(* IEC 61131-3 sources: fse/dataset/original (part 9) *)

(* ---- lb_claude_assisted_602fedacb1c4_0031.st ---- *)
PROGRAM JamDetection

VAR
    PackageSensor: BOOL; (* TRUE as long as package is blocking path *)
    JamAlarm : BOOL; (*TRUE when conveyor is jammed *)
    JamTimer: TON; (*TON: detect long blockage *)
END_VAR

JamTimer(IN:= PackageSensor, PT := T#5s);

IF JamTimer.Q = TRUE THEN
    JamAlarm := TRUE;
ELSE
    JamAlarm := FALSE;
END_IF;

END_PROGRAM

(* ---- lb_claude_assisted_66b6637cc6c5_0061.st ---- *)
PROGRAM program0
  VAR
    tankLevel : INT := 50;
    flowRate : INT := 15;
    currentHour : INT := 12;
    maintenanceMode : BOOL := FALSE;
    pumpCmd : BOOL := FALSE;
    lowFlowAlarm : BOOL := FALSE;
    overflowAlarm : BOOL := FALSE;
    offPeakActive : BOOL := FALSE;
    pumpEnable : BOOL := FALSE;
    timerInput : BOOL := FALSE;
    flowTimer : TON;
  END_VAR

  (* Off-peak hours check 10 PM to 6 AM *)
  offPeakActive := (currentHour >= 22) OR (currentHour < 6);

  (* Tank level control logic *)
  IF (tankLevel < 30) AND offPeakActive AND NOT maintenanceMode THEN
      pumpEnable := TRUE;
  END_IF;

  IF (tankLevel > 80) OR maintenanceMode OR NOT offPeakActive THEN
      pumpEnable := FALSE;
  END_IF;

  (* Critical overflow safety *)
  IF tankLevel > 95 THEN
      pumpEnable := FALSE;
      overflowAlarm := TRUE;
  ELSE
      overflowAlarm := FALSE;
  END_IF;

  (* Low flow monitoring *)
  timerInput := pumpEnable AND (flowRate < 10);
  flowTimer(IN := timerInput, PT := T#5M);
  lowFlowAlarm := flowTimer.Q;

  (* Final pump command *)
  pumpCmd := pumpEnable AND NOT overflowAlarm AND NOT maintenanceMode;
END_PROGRAM

CONFIGURATION Config0

  RESOURCE Res0 ON PLC
    TASK task0(INTERVAL := T#20ms,PRIORITY := 0);
    PROGRAM instance0 WITH task0 : program0;
  END_RESOURCE
END_CONFIGURATION

(* ---- lb_claude_assisted_6b9578db113e_0003.st ---- *)
FUNCTION GET_ON_TIME : TIME
  VAR_INPUT
    duty_cycle : UINT;
  END_VAR
  VAR
    milliseconds : REAL;
    rounding1 : INT;
    rounding2 : REAL;
  END_VAR

  milliseconds := 2.0 / 100.0 * UINT_TO_REAL(duty_cycle);

  (* get all individual unit values *)
  rounding1 := REAL_TO_INT(milliseconds * 100.0);
  rounding2 := INT_TO_REAL(rounding1) / 100000.0;

  (* create string of a real number 2 decimal places *)
  GET_ON_TIME := REAL_TO_TIME(rounding2);
END_FUNCTION

FUNCTION GET_OFF_TIME : TIME
  VAR_INPUT
    duty_cycle : UINT;
  END_VAR
  VAR
    milliseconds : REAL;
    rounding1 : INT;
    rounding2 : REAL;
  END_VAR

  milliseconds := 2.0 - (2.0 / 100.0 * UINT_TO_REAL(duty_cycle));

  (* get all individual unit values *)
  rounding1 := REAL_TO_INT(milliseconds * 100.0);
  rounding2 := INT_TO_REAL(rounding1) / 100000.0;

  (* create string of a real number 2 decimal places *)
  GET_OFF_TIME := REAL_TO_TIME(rounding2);
END_FUNCTION

PROGRAM motor_driver
  VAR
    led AT %QX0.3 : BOOL := true;
  END_VAR
  VAR
    led_on_timer : TON;
    led_off_timer : TOF;
    output_on_timer : TON;
    output_off_timer : TOF;
    input_angle : INT := 90;
    real_angle : REAL := 90.0;
    duty_cycle : UINT := 50;
    on_PT : TIME := T#2ms;
    off_PT : TIME := T#2ms;
  END_VAR
  VAR
    output_pin AT %QW1 : UINT := 65535;
  END_VAR

  (* Blink the builtin LED *)
  led_on_timer(IN := NOT(led_off_timer.Q), PT := T#50ms);
  led_off_timer(IN := led_on_timer.Q, PT := T#50ms);
  led := led_off_timer.Q;

  (* validate the servo angle *)
  IF(input_angle < 0) THEN
    input_angle := 0;

  ELSIF(input_angle > 180) THEN
    input_angle := 180;

  END_IF;

  (* control the servo *)
  real_angle := INT_TO_REAL(input_angle);
  duty_cycle := REAL_TO_UINT(100.0 / 180.0 * real_angle);

  on_PT := GET_ON_TIME(duty_cycle);
  off_PT := GET_OFF_TIME(duty_cycle);

  output_on_timer(IN := NOT(output_off_timer.Q), PT := on_PT);
  output_off_timer(IN := output_on_timer.Q, PT := off_PT);

  IF output_on_timer.Q THEN
    output_pin := 65535;

  ELSE
    output_pin := 0;

  END_IF;
END_PROGRAM

CONFIGURATION Config0

  RESOURCE Res0 ON PLC
    TASK task0(INTERVAL := T#1ms,PRIORITY := 0);
    PROGRAM instance0 WITH task0 : motor_driver;
  END_RESOURCE
END_CONFIGURATION

(* ---- lb_claude_assisted_71c3fd7363b1_0035.st ---- *)
PROGRAM Paletizador
  VAR
    Inicio AT %IX100.0 : BOOL;
    Paro AT %IX100.1 : BOOL;
    Motor_cinta_Horizontal AT %QX100.0 : BOOL;
    Motor_cinta_Inclinado AT %QX100.1 : BOOL;
    Motor_cinta_Paletizador AT %QX100.2 : BOOL;
    Contador_Cajas AT %IX100.2 : BOOL;
    Piston_1 AT %QX100.3 : BOOL;
    Sensor_Piston_1 AT %IX100.3 : BOOL;
  END_VAR
  VAR
    CTU0 : CTU;
  END_VAR
  VAR
    Piston_Compuerta AT %QX100.4 : BOOL;
    Sensor_Piston_Compuerta AT %IX100.4 : BOOL;
    Compuerta AT %QX100.5 : BOOL;
    Sensor_Compuerta AT %IX100.5 : BOOL;
  END_VAR
  VAR
    CTU1 : CTU;
  END_VAR
  VAR
    Generador_Cajas AT %QX100.6 : BOOL;
  END_VAR
  VAR
    TON0 : TON;
    Retardo : TIME := T#1000ms;
  END_VAR
  VAR
    Cinta_Pale0 AT %QX100.7 : BOOL;
    Cinta_Pale1 AT %QX100.8 : BOOL;
    Generador_pales AT %QX100.9 : BOOL;
    Cinta_Paletizador AT %QX100.10 : BOOL;
    Sensor_Pale_0 AT %IX100.6 : BOOL;
    Sensor_Pale_1 AT %IX100.7 : BOOL;
    limite_altura AT %QX100.12 : BOOL;
    subir_pale AT %QX100.11 : BOOL;
    bajar_pale AT %QX100.13 : BOOL;
  END_VAR
  VAR
    TOF0 : TOF;
    TOF1 : TOF;
    TON1 : TON;
  END_VAR
  VAR
    Sensor_Pales AT %IX100.8 : BOOL;
    sensor_ascensor AT %IX100.9 : BOOL;
  END_VAR
  VAR
    CTU2 : CTU;
    TON2 : TON;
  END_VAR
  VAR
    sensor_bajada AT %IX100.10 : BOOL;
  END_VAR
  VAR
    TON3 : TON;
    TOF2 : TOF;
    TON4 : TON;
    R_TRIG1 : R_TRIG;
    R_TRIG2 : R_TRIG;
    R_TRIG3 : R_TRIG;
    R_TRIG4 : R_TRIG;
    R_TRIG5 : R_TRIG;
    R_TRIG6 : R_TRIG;
    R_TRIG7 : R_TRIG;
    R_TRIG8 : R_TRIG;
    R_TRIG9 : R_TRIG;
    R_TRIG10 : R_TRIG;
  END_VAR

  Motor_cinta_Horizontal := NOT(Paro) AND (Generador_Cajas OR Inicio OR Motor_cinta_Horizontal OR Motor_cinta_Inclinado OR Motor_cinta_Paletizador);
  Motor_cinta_Inclinado := NOT(Paro) AND (Generador_Cajas OR Inicio OR Motor_cinta_Horizontal OR Motor_cinta_Inclinado OR Motor_cinta_Paletizador);
  Motor_cinta_Paletizador := NOT(Paro) AND (Generador_Cajas OR Inicio OR Motor_cinta_Horizontal OR Motor_cinta_Inclinado OR Motor_cinta_Paletizador);
  R_TRIG1(CLK := Contador_Cajas);
  R_TRIG2(CLK := Sensor_Piston_1);
  CTU0(CU := R_TRIG1.Q, R := R_TRIG2.Q, PV := 2);
  Piston_1 := CTU0.Q;
  R_TRIG3(CLK := Contador_Cajas);
  CTU1(CU := R_TRIG3.Q, R := Sensor_Piston_Compuerta, PV := 6);
  TON0(IN := CTU1.Q, PT := Retardo);
  Piston_Compuerta := TON0.Q;
  Sensor_Piston_Compuerta := Sensor_Piston_Compuerta;
  Generador_Cajas := NOT(Paro) AND (Generador_Cajas OR Inicio OR Motor_cinta_Horizontal OR Motor_cinta_Inclinado OR Motor_cinta_Paletizador);
  Sensor_Piston_1 := NOT(NOT(Sensor_Piston_1));
  TOF1(IN := Sensor_Piston_Compuerta, PT := T#3500ms);
  Compuerta := TOF1.Q;
  TON1(IN := Sensor_Pales, PT := T#2000ms);
  TOF0(IN := TON1.Q, PT := T#3500ms);
  subir_pale := TOF0.Q;
  limite_altura := TOF0.Q;
  bajar_pale := Compuerta;
  R_TRIG4(CLK := sensor_ascensor);
  TON3(IN := sensor_bajada, PT := T#2000ms);
  CTU2(CU := R_TRIG4.Q, R := TON3.Q, PV := 3);
  TON2(IN := CTU2.Q, PT := T#2000ms);
  IF TON2.Q THEN
    limite_altura := TRUE; (*set*)
  END_IF;
  IF TON2.Q THEN
    bajar_pale := TRUE; (*set*)
  END_IF;
  R_TRIG5(CLK := sensor_bajada);
  Cinta_Pale0 := NOT(Paro) AND (Cinta_Pale0 OR Cinta_Pale1 OR Cinta_Paletizador OR Generador_pales OR Inicio OR sensor_ascensor AND R_TRIG5.Q);
  R_TRIG6(CLK := sensor_bajada);
  Cinta_Pale1 := NOT(Paro) AND (Cinta_Pale0 OR Cinta_Pale1 OR Cinta_Paletizador OR Generador_pales OR Inicio OR sensor_ascensor AND R_TRIG6.Q);
  R_TRIG7(CLK := sensor_bajada);
  Cinta_Paletizador := NOT(Paro) AND (Cinta_Pale0 OR Cinta_Pale1 OR Cinta_Paletizador OR Generador_pales OR Inicio OR sensor_ascensor AND R_TRIG7.Q);
  R_TRIG8(CLK := sensor_bajada);
  Generador_pales := NOT(Paro) AND (Cinta_Pale0 OR Cinta_Pale1 OR Cinta_Paletizador OR Generador_pales OR Inicio OR sensor_ascensor AND R_TRIG8.Q);
  TOF2(IN := Sensor_Pales, PT := T#3700ms);
  TON4(IN := TOF2.Q, PT := T#3700ms);
  IF TON4.Q THEN
    Cinta_Pale0 := FALSE; (*reset*)
  END_IF;
  IF TON4.Q THEN
    Cinta_Pale1 := FALSE; (*reset*)
  END_IF;
  IF TON4.Q THEN
    Cinta_Paletizador := FALSE; (*reset*)
  END_IF;
  IF TON4.Q THEN
    Generador_pales := FALSE; (*reset*)
  END_IF;
  R_TRIG9(CLK := sensor_bajada);
  IF NOT(Paro) AND (Cinta_Pale0 OR Cinta_Pale1 OR Cinta_Paletizador OR Generador_pales OR Inicio OR sensor_ascensor AND R_TRIG9.Q) THEN
    limite_altura := FALSE; (*reset*)
  END_IF;
  R_TRIG10(CLK := sensor_bajada);
  IF NOT(Paro) AND (Cinta_Pale0 OR Cinta_Pale1 OR Cinta_Paletizador OR Generador_pales OR Inicio OR sensor_ascensor AND R_TRIG10.Q) THEN
    bajar_pale := FALSE; (*reset*)
  END_IF;
END_PROGRAM

CONFIGURATION Config0

  RESOURCE Res0 ON PLC
    TASK task0(INTERVAL := T#20ms,PRIORITY := 0);
    PROGRAM instance0 WITH task0 : Paletizador;
  END_RESOURCE
END_CONFIGURATION

(* ---- lb_claude_assisted_7966a27f0066_0051.st ---- *)
PROGRAM MAIN
  VAR
    Input_I1_S0Powermeter AT %IX0.0 : BOOL;
    Input_I2_LightSwitch AT %IX0.1 : BOOL;
    Input_I3_EstopNO AT %IX0.2 : BOOL;
    Input_I4_EstopNC AT %IX0.3 : BOOL;
    Input_I5_ToggleLeft AT %IX0.4 : BOOL;
    Input_I6_ToggleRight AT %IX0.5 : BOOL;
    Input_I7_ButtonGreen AT %IX0.6 : BOOL;
    Input_I8_ButtonRed AT %IX0.7 : BOOL;
    Output_Q1_230vLight AT %QX0.0 : BOOL;
    Output_Q2 AT %QX0.1 : BOOL;
    Output_Q3_StacklightGreen AT %QX0.2 : BOOL;
    Output_Q4_StacklightYellow AT %QX0.3 : BOOL;
    Output_Q5_StacklightRed AT %QX0.4 : BOOL;
    Output_Q6 AT %QX0.5 : BOOL;
    Output_Q7 AT %QX0.6 : BOOL;
    Output_Q8 AT %QX0.7 : BOOL;
    PWM_0_LED1 AT %QW0 : UINT;
    PWM_1_LED2 AT %QW1 : UINT;
    ModIO_Q1 AT %QX100.0 : BOOL;
    ModIO_Q2 AT %QX100.1 : BOOL;
    ModIO_Q3 AT %QX100.2 : BOOL;
    ModIO_Q4 AT %QX100.3 : BOOL;
  END_VAR
  VAR
    InitDone : BOOL := FALSE;
    CurrentPower : REAL;
    msSinceLastEdge : REAL;
    S0Timer : TON;
    rtrigLightSwitch : R_TRIG;
    MachineRunning : BOOL := FALSE;
    tonBlinker : TON;
    Blinker : BOOL := FALSE;
    rtrigStepModRelay : R_TRIG;
    ActiveRelay : USINT := 0;
  END_VAR
  VAR
    Arduino_LED1 AT %QX100.4 : BOOL := 0;
    Arduino_LED2 AT %QX100.5 : BOOL := 0;
    Arduino_LED3 AT %QX100.6 : BOOL := 0;
    Arduino_LED4 AT %QX100.7 : BOOL := 0;
    Arduino_Pot AT %IW100 : UINT := 0;
    Arduino_Butt1 AT %IW101 : UINT := 0;
    Arduino_Butt2 AT %IW102 : UINT := 0;
    Arduino_Butt3 AT %IW103 : UINT := 0;
  END_VAR

  (* This is a testing program to test most functions on a PiPLC                                      *)
  (* Make sure to activate the "Binary-6 PiPLC" hardware layer on your PLC before uploading this code *)

  IF NOT InitDone THEN
    (* Oneshots at init *)

    (* Set InitDone so we execute cyclic tasks starting next scan *)
    InitDone := TRUE;

  ELSE
    (*----------------------------------------*)
    (* Cyclic calls after init oneshots       *)
    (*----------------------------------------*)
    (* Global blinker *)
    tonBlinker(IN := NOT tonBlinker.Q, PT := T#500ms);
    IF tonBlinker.Q THEN
      Blinker := NOT Blinker;
    END_IF;

    (* "Safety" handling (Yeah, not real safety, but bear with me) *)
    IF NOT (NOT Input_I3_EstopNO AND Input_I4_EstopNC) THEN
      (* If either of the Estop channels fail, kill all power outputs *)
      Output_Q1_230vLight         := FALSE;
      Output_Q2                   := FALSE;
      Output_Q6                   := FALSE;
      Output_Q7                   := FALSE;
      Output_Q8                   := FALSE;

      ModIO_Q1        := FALSE;
      ModIO_Q2        := FALSE;
      ModIO_Q3        := FALSE;
      ModIO_Q4        := FALSE;

      Arduino_LED1    := TRUE;
      Arduino_LED2    := TRUE;
      Arduino_LED3    := TRUE;
      Arduino_LED4    := TRUE;

      PWM_0_LED1      := 0;
      PWM_1_LED2      := 0;

      ActiveRelay     := 0;
      MachineRunning  := FALSE;

      (* Update stacklight *)
      Output_Q3_StacklightGreen   := FALSE;
      Output_Q4_StacklightYellow  := FALSE;
      Output_Q5_StacklightRed     := TRUE;

    ELSE
      (* As long as Estop is good, execute regular logic *)

      (* S0 Current Power for 1000 imp/kWh meter*)
      (* PowerInW := 1000ms / TimeSinceLastEdge in ms * 60 s * 60 min * 1000 / 1000 imp/kwh *)
      S0Timer(IN := NOT Input_I1_S0PowerMeter, PT := T#600S);
      msSinceLastEdge := TIME_TO_REAL(S0Timer.ET);
      CurrentPower := 1000.0 / msSinceLastEdge * 3600.0;

      (* Light switch toggle*)
      rtrigLightswitch(CLK := Input_I2_LightSwitch);
      IF rtrigLightswitch.Q THEN
        Output_Q1_230vLight := NOT Output_Q1_230vLight;
      END_IF;

      (*----------------------------------------*)
      (* Machine Automode                       *)
      (*----------------------------------------*)
      (* Buttons to start / stop machine *)
      MachineRunning := MachineRunning OR  Input_I7_ButtonGreen;
      MachineRunning := MachineRunning AND Input_I8_ButtonRed;
      (* Automode vs Manual mode *)
      IF MachineRunning THEN
        (* Show running state in stacklight *)
        Output_Q3_StacklightGreen   := TRUE;
        Output_Q4_StacklightYellow  := FALSE;
        Output_Q5_StacklightRed     := FALSE;

        (* Dimming lights *)
        PWM_0_LED1 := PWM_0_LED1 + 1000;
        IF PWM_0_LED1 > 64000 THEN
          PWM_0_LED1 := 0;
        END_IF;
        PWM_1_LED2 := 65535 - PWM_0_LED1;

        (* Modbus IO *)
        rtrigStepModRelay(CLK := Blinker);
        IF rtrigStepModRelay.Q THEN

          ActiveRelay := ActiveRelay + 1;

          IF ActiveRelay > 4 THEN
            ActiveRelay := 1;
          END_IF;

          ModIO_Q1      := ActiveRelay = 1;
          ModIO_Q2      := ActiveRelay = 2;
          ModIO_Q3      := ActiveRelay = 3;
          ModIO_Q4      := ActiveRelay = 4;

          Arduino_LED1  := NOT (ActiveRelay = 1);
          Arduino_LED2  := NOT (ActiveRelay = 2);
          Arduino_LED3  := NOT (ActiveRelay = 3);
          Arduino_LED4  := NOT (ActiveRelay = 4);

        END_IF;

        (* 1-Wire temp probe *)

        (* Arduino Slave *)

        (* I²C Servos *)

        (* EtherCAT *)

      ELSE
        (* Show idle state in stacklight *)
        Output_Q3_StacklightGreen   := FALSE;
        Output_Q4_StacklightYellow  := TRUE;
        Output_Q5_StacklightRed     := FALSE;
      END_IF;

    END_IF;

  END_IF;
END_PROGRAM

CONFIGURATION Config0

  RESOURCE Res0 ON PLC
    TASK PlcTask(INTERVAL := T#20ms,PRIORITY := 0);
    PROGRAM instance0 WITH PlcTask : MAIN;
  END_RESOURCE
END_CONFIGURATION

(* ---- lb_claude_assisted_876e5799c2c7_0075.st ---- *)
PROGRAM AutomatedReactorControl
VAR
    reactorMode AT %IW0.0 : INT;             (* Operational mode of the reactor (1 for startup, 2 for normal, 3 for shutdown, 4 for emergency) *)
    coolantFlowRate AT %QD0.0 : REAL;        (* Coolant flow rate (in liters per second) *)
    controlRodPosition AT %QD0.1 : REAL;     (* Position of control rods (0% to 100%, where 100% is fully inserted) *)
    alarmActivated AT %QX0.0 : BOOL;         (* State of the alarm system *)
END_VAR

(* Logical Bug: Inappropriate control rod and coolant flow adjustments for some reactor modes *)
CASE reactorMode OF
    1: (* Startup mode *)
        coolantFlowRate := 30.0;   (* Moderate coolant flow *)
        controlRodPosition := 20.0; (* Partially withdrawn control rods *)
    2: (* Normal operation mode *)
        coolantFlowRate := 50.0;   (* High coolant flow *)
        controlRodPosition := 50.0; (* Halfway inserted control rods *)
    3: (* Shutdown mode *)
        coolantFlowRate := 20.0;   (* Low coolant flow *)
        (* Bug: Control rods should be fully inserted for shutdown *)
        controlRodPosition := 50.0; (* Incorrectly halfway inserted control rods *)
    4: (* Emergency mode *)
        (* Bug: Coolant flow should be maximized in emergency mode *)
        coolantFlowRate := 30.0;   (* Insufficient coolant flow for emergency *)
        controlRodPosition := 100.0; (* Fully inserted control rods *)
        (* ActivateAlarm(); *)
        alarmActivated := TRUE;
    ELSE
        (* Default safe state in case of an unrecognized mode *)
        (* ActivateAlarm(); *)
        alarmActivated := TRUE;
        coolantFlowRate := 0.0;
        controlRodPosition := 100.0; (* Fully insert control rods *)
END_CASE;

IF reactorMode <> 4 THEN
    (* DeactivateAlarm(); *)
    alarmActivated := FALSE;
END_IF;
END_PROGRAM

CONFIGURATION STD_CONF

  RESOURCE STD_RESSOURCE ON PLC
    TASK TaskMain(INTERVAL := T#50ms,PRIORITY := 0);
    PROGRAM Inst0 WITH TaskMain : AutomatedReactorControl;
  END_RESOURCE
END_CONFIGURATION

(* ---- lb_claude_assisted_895a3a5527b4_0023.st ---- *)
PROGRAM Mixing
  VAR
    m AT %QX0.0 : BOOL;
    a AT %QX0.1 : BOOL;
    b AT %QX0.2 : BOOL;
    d1 AT %QX0.3 : BOOL;
    d2 AT %QX0.4 : BOOL;
    e1 AT %QX0.5 : BOOL;
    e2 AT %QX0.6 : BOOL;
    f AT %QX0.7 : BOOL;
    g AT %QX1.0 : BOOL;
    l AT %QX1.1 : BOOL;
    EA AT %QX2.0 : BOOL;
    EB AT %QX2.1 : BOOL;
    ED AT %QX2.2 : BOOL;
    EE AT %QX2.3 : BOOL;
    EF AT %QX2.4 : BOOL;
    EG AT %QX2.5 : BOOL;
    M1 AT %QX2.6 : BOOL;
    M2 AT %QX2.7 : BOOL;
    X0 AT %QX3.0 : BOOL := TRUE;
    X1 AT %QX3.1 : BOOL;
    X2 AT %QX3.2 : BOOL;
    X3 AT %QX3.3 : BOOL;
    X4 AT %QX3.4 : BOOL;
    X5 AT %QX3.5 : BOOL;
    X6 AT %QX3.6 : BOOL;
    X7 AT %QX3.7 : BOOL;
    X8 AT %QX4.0 : BOOL;
    T0 AT %QX5.0 : BOOL;
    T1 AT %QX5.1 : BOOL;
    T2 AT %QX5.2 : BOOL;
    T3 AT %QX5.3 : BOOL;
    T4 AT %QX5.4 : BOOL;
    T5 AT %QX5.5 : BOOL;
    T6 AT %QX5.6 : BOOL := FALSE;
    T7 AT %QX5.7 : BOOL := FALSE;
    T8 AT %QX6.0 : BOOL := FALSE;
    PV AT %QW0 : INT := 3;
    CV AT %QW1 : INT;
    time_1 AT %QW2 : INT := 0;
    time_2 AT %QW3 : INT := 0;
    timer_gauge_1 AT %QW4 : INT := 5;
    timer_gauge_2 AT %QW5 : INT := 5;
    CU AT %QX7.0 : BOOL := TRUE;
  END_VAR
  VAR
    TP1 : TP;
    TP2 : TP;
    CTU0 : CTU;
    TON0 : TON;
    _TMP_INT_TO_TIME191_OUT : TIME;
    _TMP_INT_TO_TIME42_OUT : TIME;
    R_TRIG1 : R_TRIG;
    _TMP_INT_TO_TIME43_OUT : TIME;
    _TMP_TIME_TO_INT188_OUT : INT;
    _TMP_TIME_TO_INT40_OUT : INT;
  END_VAR

  T0 := m AND X0;
  T1 := d1 AND X1;
  T2 := a AND X2;
  T3 := e1 AND X4;
  T4 := b AND X5;
  T5 := e2 AND d2 AND X6 AND X3;
  IF T0 THEN
    X0 := FALSE; (*reset*)
  END_IF;
  IF T0 THEN
    X1 := TRUE; (*set*)
  END_IF;
  IF T0 THEN
    X4 := TRUE; (*set*)
  END_IF;
  IF T1 THEN
    X1 := FALSE; (*reset*)
  END_IF;
  IF T1 THEN
    X2 := TRUE; (*set*)
  END_IF;
  IF T2 THEN
    X2 := FALSE; (*reset*)
  END_IF;
  IF T2 THEN
    X3 := TRUE; (*set*)
  END_IF;
  IF T3 THEN
    X4 := FALSE; (*reset*)
  END_IF;
  IF T3 THEN
    X5 := TRUE; (*set*)
  END_IF;
  IF T4 THEN
    X5 := FALSE; (*reset*)
  END_IF;
  IF T4 THEN
    X6 := TRUE; (*set*)
  END_IF;
  IF T5 THEN
    X3 := FALSE; (*reset*)
  END_IF;
  IF T5 THEN
    X6 := FALSE; (*reset*)
  END_IF;
  IF T6 THEN
    X7 := FALSE; (*reset*)
  END_IF;
  IF T6 THEN
    X8 := TRUE; (*set*)
  END_IF;
  EA := X1;
  ED := X3;
  EB := X4;
  EE := X6;
  EF := X7;
  _TMP_INT_TO_TIME191_OUT := INT_TO_TIME(timer_gauge_2);
  TP2(IN := X8, PT := _TMP_INT_TO_TIME191_OUT);
  M2 := TP2.Q;
  _TMP_INT_TO_TIME42_OUT := INT_TO_TIME(timer_gauge_1);
  TP1(IN := X7, PT := _TMP_INT_TO_TIME42_OUT);
  M1 := TP1.Q;
  EG := X8;
  R_TRIG1(CLK := X8 AND CU);
  CTU0(CU := R_TRIG1.Q, R := T8, PV := PV);
  _TMP_INT_TO_TIME43_OUT := INT_TO_TIME(timer_gauge_2);
  TON0(IN := CTU0.Q, PT := _TMP_INT_TO_TIME43_OUT);
  T8 := TON0.Q;
  CV := CTU0.CV;
  T6 := l AND f AND X7;
  IF T5 THEN
    X7 := TRUE; (*set*)
  END_IF;
  IF T7 THEN
    X8 := FALSE; (*reset*)
  END_IF;
  IF T7 THEN
    X7 := TRUE; (*set*)
  END_IF;
  IF T8 THEN
    X8 := FALSE; (*reset*)
  END_IF;
  IF T8 THEN
    X0 := TRUE; (*set*)
  END_IF;
  T7 := g AND X8;
  _TMP_TIME_TO_INT188_OUT := TIME_TO_INT(TP1.ET);
  time_1 := _TMP_TIME_TO_INT188_OUT;
  _TMP_TIME_TO_INT40_OUT := TIME_TO_INT(TP2.ET);
  time_2 := _TMP_TIME_TO_INT40_OUT;
END_PROGRAM

CONFIGURATION Config0

  RESOURCE Res0 ON PLC
    TASK task0(INTERVAL := T#20ms,PRIORITY := 0);
    PROGRAM instance0 WITH task0 : Mixing;
  END_RESOURCE
END_CONFIGURATION

(* ---- lb_claude_assisted_97f2e223644e_0009.st ---- *)
TYPE
  SuperStatesEnum : (ST_INICIALIZACE, ST_RESET_POSITION_OF_MOTORS, ST_WAIT_FOR_COMMAND, ST_MODE_SELECTION, ST_MANUAL_MODE, ST_AUTOMATIC_MODE, ST_CHECK_POSITION_OF_MOTORS, ST_STOP, ST_EMERGENCY_STOP) := ST_INICIALIZACE;
END_TYPE

PROGRAM SuperStavy
  VAR
    I_Start AT %IX0.6 : BOOL := 0;
    Start_RTRIG AT %IX0.7 : BOOL := 1;
    I_PowerOn AT %IX1.1 : BOOL := 1;
    I_StopBtn AT %IX1.2 : BOOL;
    I_StopResBtn AT %IX1.3 : BOOL;
    I_EmStopBtn AT %IX1.4 : BOOL;
    I_EmStopResBtn AT %IX1.5 : BOOL;
    I_ManualSelector AT %IX1.6 : BOOL;
    I_AutomaticSelector AT %IX1.7 : BOOL := 1;
  END_VAR
  VAR
    SuperStates : SuperStatesEnum := ST_INICIALIZACE;
  END_VAR
  VAR
    I_A0 AT %IX0.0 : BOOL;
    I_A1 AT %IX0.1 : BOOL;
    I_B0 AT %IX0.2 : BOOL;
    I_B1 AT %IX0.3 : BOOL;
    I_C0 AT %IX0.4 : BOOL;
    I_C1 AT %IX0.5 : BOOL;
  END_VAR
  VAR
    I_Qt : BOOL;
  END_VAR
  VAR
    Q_A AT %QX0.4 : BOOL;
    Q_B AT %QX0.5 : BOOL;
    Q_C AT %QX0.6 : BOOL;
  END_VAR
  VAR
    Q_PositionOk : BOOL;
    Q_PositionNotOk : BOOL;
    Q_It : BOOL;
    InputArr : ARRAY [0..7] OF BYTE;
    InputWord : INT;
    TRANS_MATX : ARRAY [0..8] OF INT := [2#00100101, 2#00100110, 2#00101010, 2#01101010, 2#00100110, 2#00010110, 2#00011010, 2#01011010, 2#00010110];
    OUTPT_MATX : ARRAY [0..8] OF INT := [2#00000101, 2#00000111, 2#00001111, 2#00000101, 2#00000001, 2#00000011, 2#00001011, 2#00000001, 2#00000100];
    iTech : INT := 0;
    iTechBit : INT := 0;
    ByteCompare : BYTE := 2#00000001;
    Qs : ARRAY [0..7] OF BOOL;
    TechnologicalSequenceState : INT := 0;
    SuperSequenceState : INT;
    TON_0 : TON;
    BlastingTime : TIME := t#5s;
  END_VAR

  IF (I_EMSTOPBTN = true) THEN

        SuperStates := ST_EMERGENCY_STOP;

    END_IF;

    CASE SuperStates OF

      ST_INICIALIZACE:
        SuperSequenceState := 1;
        IF (I_Start = true) (*AND (I_PowerOn = true)*) THEN (*Uprava 10.11.2021*)

          SuperStates := ST_RESET_POSITION_OF_MOTORS;

        END_IF;

      ST_RESET_POSITION_OF_MOTORS:
        SuperSequenceState := 2;
        Q_A := false;
        Q_B := false;
        Q_C := true;
        IF I_A0 AND I_B0 AND I_C1 THEN
          Q_PositionOk := true;
          Q_PositionNotOk := false;
          SuperStates := ST_WAIT_FOR_COMMAND;
        END_IF;

      ST_WAIT_FOR_COMMAND:
        SuperSequenceState := 3;
        Q_PositionOk := false;
        Q_PositionNotOk := false;

        SuperStates := ST_MODE_SELECTION;

      ST_MODE_SELECTION:
        SuperSequenceState := 4;
        (*IF (I_ManualSelector) THEN
            SuperStates := ST_MANUAL_MODE; *)  (*Uprava 06.05.2021*)
        (*ELSIF (I_AutomaticSelector) THEN *)
            SuperStates := ST_AUTOMATIC_MODE;
        (*END_IF;*)    (*Uprava 06.05.2021*)
        (*TODO// Comeback from this state to STOP*)

      ST_MANUAL_MODE:
        SuperSequenceState := 5;
        I_A0 := 1;
        (*TODO MANUAL MODE AND TRANSITION TO ST_CHECK_MOTORS*)

      ST_AUTOMATIC_MODE:
        SuperSequenceState := 6;

        (*  Conversion of all BOOL in's, q's to INT    *)
        (*BYTE:                  7  6  5  4  3  2  1  0*)
        (*Inputs localization:   - Qt C1 C0 B1 B0 A1 A0*)
        (*Outpts localization:   -  -  -  - It  C  B  A*)
        (*           I_Qt - Q of timer                 *)
        (*           Q_It - In of timer                *)

        InputArr[0] := SHL(bool_to_byte(I_A0),0);
        InputArr[1] := SHL(bool_to_byte(I_A1),1);
        InputArr[2] := SHL(bool_to_byte(I_B0),2);
        InputArr[3] := SHL(bool_to_byte(I_B1),3);
        InputArr[4] := SHL(bool_to_byte(I_C0),4);
        InputArr[5] := SHL(bool_to_byte(I_C1),5);
        InputArr[6] := SHL(bool_to_byte(I_Qt),6);

        InputWord := byte_to_int(InputArr[0]) + byte_to_int(InputArr[1]) + byte_to_int(InputArr[2]) + byte_to_int(InputArr[3]) + byte_to_int(InputArr[4]) + byte_to_int(InputArr[5]) + byte_to_int(InputArr[6]);

        (*   End of Conversion   *)

        IF (InputWord = TRANS_MATX[iTech]) THEN

          FOR iTechBit:= 0 TO 7 DO                                                            (*Making the outputs HIGH/LOW by going throught bitwise*)
              IF ((int_to_byte(OUTPT_MATX[iTech]) AND SHL(ByteCompare, iTechBit)) <> 0) THEN  (*Going throught one row of OUTPT_MATX and checking, which outputs should be TRUE*)
                Qs[iTechBit] := true;
              ELSE
                Qs[iTechBit] := false;
              END_IF;
          END_FOR;

          (*Mapping of outputs*)
          Q_A := Qs[0];
          Q_B := Qs[1];
          Q_C := Qs[2];
          Q_It := Qs[3];
          (*End of mapping of outputs*)

          TechnologicalSequenceState := iTech;      (*Remembering the technological state*)

          iTech := iTech + 1;                       (*Going to the next state*)

        END_IF;

        (*Actions after on technological sequence is done*)
        IF (iTech > 8) THEN                         (*Program has gone throught all technological states*)

          iTech := 0;                               (*Reset sequence*)
        END_IF;

       (*ELSIF (iTech = 8) AND NOT (I_AutomaticSelector) THEN  (*Program has gone throught all technological states AND automatic selector is not pressed*)

        (*  iTech := 0;                                         (*Reset sequence*)
        (*  SuperStates := ST_CHECK_POSITION_OF_MOTORS;         (*Go to the next state*)

        (*ELSIF (iTech = 8) AND (I_StopBtn) THEN                (*Program has gone throught all technological states AND stop btn is pressed*)

         (* SuperStates := ST_STOP;                               (*Go to stop state*)

       (* END_IF;*)

      ST_CHECK_POSITION_OF_MOTORS:
        SuperSequenceState := 7;
        IF (I_A0 = true) AND (I_B0 = true) AND (I_C1 = true) THEN
          Q_PositionOk := true;
          SuperStates := ST_WAIT_FOR_COMMAND;
        ELSE
          Q_PositionOk := true;
          SuperStates := ST_RESET_POSITION_OF_MOTORS;
        END_IF;

      ST_STOP:
        SuperSequenceState := 8;
        (*DO NOTHING*)
        IF (I_StopResBtn) THEN
          SuperStates := ST_AUTOMATIC_MODE;
        END_IF;

      ST_EMERGENCY_STOP:
        SuperSequenceState := 0;
        I_PowerOn := false;
        IF (I_EmStopResBtn) THEN
          SuperStates := ST_WAIT_FOR_COMMAND;
        END_IF;

    END_CASE;

    (*Function block calling*)

    TON_0(IN := I_B1, PT := BlastingTime, Q => I_Qt);

    (*End of Function block calling*)
END_PROGRAM

CONFIGURATION Config0

  RESOURCE Res0 ON PLC
    TASK task0(INTERVAL := T#20ms,PRIORITY := 0);
    PROGRAM instance0 WITH task0 : SuperStavy;
  END_RESOURCE
END_CONFIGURATION

(* ---- lb_claude_assisted_a6650ce22d1a_0020.st ---- *)
PROGRAM Gate_Controller
  VAR
    Start_Loop : BOOL := False;
    one_hour : TIME := T#1h;
    One_Hour_Timer : TON;
    Gate_Open : BOOL := False;
  END_VAR
  VAR_OUTPUT
    Close_Gate_Inst : BOOL := False;
  END_VAR
  VAR_INPUT
    Sensed_Car : BOOL := False;
    Sensed_Car_Inst : BOOL := False;
    Sensed_App : BOOL := False;
    Mobile_Inst : BOOL := False;
    Mobile_Auth : STRING;
  END_VAR
  VAR
    my_defined_str : STRING := '"1234"';
  END_VAR

  One_Hour_Timer(IN := NOT(Start_Loop), PT := one_hour);

  IF One_Hour_Timer.Q THEN
    IF Gate_Open THEN
      Close_Gate_Inst := True;
      Gate_Open := False;
    END_IF;
  END_IF;

  IF Sensed_App THEN
    (* How can I do some authentication here? *)
    IF EQ(Mobile_Auth, my_defined_str) THEN
      Close_Gate_Inst := XOR(Mobile_Inst, Gate_Open);
      Gate_Open := Mobile_Inst;
    END_IF;
  END_IF;

  IF AND(Sensed_Car, Sensed_Car_Inst) THEN
    Close_Gate_Inst := XOR(Sensed_Car_Inst, Gate_Open);
    Gate_Open := Sensed_Car_Inst;
  END_IF;

  Start_Loop := One_Hour_Timer.Q;
END_PROGRAM

CONFIGURATION Config0

  RESOURCE Res0 ON PLC
    TASK task0(INTERVAL := T#20ms,PRIORITY := 0);
    PROGRAM instance0 WITH task0 : Gate_Controller;
  END_RESOURCE
END_CONFIGURATION

(* ---- lb_claude_assisted_aa88c9df37fb_0005.st ---- *)
PROGRAM cybICS
  VAR
    (* heartbeat LED on the PCB *)
    systemSen AT %MW108 : UINT := 0;
    boSen AT %MW110 : UINT := 0;
    heartbeat AT %QX0.0 : BOOL;
    compressor AT %QX0.1 : BOOL;
    systemValve AT %QX0.2 : BOOL;
    gstSig AT %QX0.3 : BOOL;
    gst AT %MW100 : UINT := 0;
    hpt AT %MW102 : UINT := 0;
    stop AT %MW104 : UINT := 0;
    manual AT %MW106 : UINT := 0;

    compressorState AT %MW200 : UINT;
    gstState AT %MW202 : UINT;
  END_VAR
  VAR
    (* Counter LED heartbeat *)
    countHeartbeat : UINT := 0;
  END_VAR

  (* System heartbeat *)
  IF countHeartbeat < 20 THEN
    heartbeat := FALSE;
  ELSIF countHeartbeat < 40 THEN
    heartbeat := TRUE;
  ELSE
    countHeartbeat := 0;
  END_IF;

  (* System running state *)
  IF stop < 1 THEN
    (* System running in automatic mode *)
    IF manual < 1 THEN
      (* Refill GST, when below 60 and fill it up to 254 *)
      IF gst < 60 AND gstState = 0 THEN
        gstState := 1;
      ELSIF gst < 240 AND gstState = 1 THEN
        gstState := 1;
      ELSE
        gstState := 0;
      END_IF;

      (* Run compressor when below 60 and fill it up to 89 *)
      (* Only run compressor, when GST > 50 *)
      IF hpt < 60 AND compressorState = 0 AND gst > 50 THEN
        compressorState := 1;
      ELSIF hpt < 90 AND compressorState = 1 AND gst > 50 THEN
        compressorState := 1;
      ELSE
        compressorState := 0;
      END_IF;

      IF hpt > 50 AND hpt<100 THEN
        systemValve := TRUE;
      ELSE
        systemValve := FALSE;
      END_IF;

      IF compressorState = 1 THEN
        compressor := TRUE;
      ELSE
        compressor := FALSE;
      END_IF;

      IF gstState = 1 THEN
        gstSig := TRUE;
      ELSE
        gstSig := FALSE;
      END_IF;
      (* ELSE System running in manual mode *)
    END_IF;
  (* System stop state *)
  ELSE
    compressorState := 0;
    compressor := FALSE;
    systemValve := FALSE;
    gstState := 0;
    gstSig := FALSE;
  END_IF;

  (* Increase the counters *)
  countHeartbeat := countHeartbeat + 1;
END_PROGRAM

CONFIGURATION Config0
  RESOURCE Res0 ON PLC
    TASK TaskMain(INTERVAL := T#50ms,PRIORITY := 0);
    PROGRAM Inst0 WITH TaskMain : cybICS;
  END_RESOURCE
END_CONFIGURATION

(* ---- lb_claude_assisted_e066873262e0_0027.st ---- *)
PROGRAM My_Program
  VAR
    button1 AT %IX0.0 : BOOL;
    button2 AT %IX0.1 : BOOL;
    led AT %QX0.0 : BOOL;
  END_VAR

  VAR
    LED_STATE : BOOL;
    ALARM_STATE: BOOL;
  END_VAR

  LED_STATE := (button1 = button2) AND (button1 = TRUE);
  ALARM_STATE := (button1 = TRUE) AND (button2 = FALSE);
  IF LED_STATE OR ALARM_STATE THEN
    led := TRUE;
  ELSE
    led := FALSE;
  END_IF;
END_PROGRAM

CONFIGURATION STD_CONF

  RESOURCE STD_RESSOURCE ON PLC
    TASK TaskMain(INTERVAL := T#50ms,PRIORITY := 0);
    PROGRAM Inst0 WITH TaskMain : My_Program;
  END_RESOURCE
END_CONFIGURATION

(* ---- lb_claude_assisted_eb6f0bbd77cb_0054.st ---- *)
PROGRAM program0
  VAR
    Inp0 AT %IX0.0 : BOOL;
    Inp1 AT %IX0.1 : BOOL;
    Inp2 AT %IX0.2 : BOOL;
    Inp3 AT %IX0.3 : BOOL;
    Inp4 AT %IX0.4 : BOOL;
    Inp5 AT %IX0.5 : BOOL;
    Inp6 AT %IX0.6 : BOOL;
    Inp7 AT %IX0.7 : BOOL;
    Ana0 AT %IW0 : UINT := 0;
    Ana1 AT %IW1 : UINT := 0;
    Out1 AT %QX0.1 : BOOL;
    Out2 AT %QX0.2 : BOOL;
    Out3 AT %QX0.3 : BOOL;
    Out4 AT %QX0.4 : BOOL;
    Out5 AT %QX0.5 : BOOL;
    Out6 AT %QX0.6 : BOOL;
    Out7 AT %QX0.7 : BOOL;
  END_VAR
  VAR
    Cval0 : INT := 0;
    Cval1 : INT := 0;
  END_VAR
  VAR
    Aout0 AT %QW0 : UINT := 60000;
    Aout3 AT %QW3 : INT;
  END_VAR
  VAR
    Cout : BOOL;
    TON0 : TON;
  END_VAR
  VAR
    Out0 AT %QX0.0 : BOOL;
  END_VAR
  VAR
    TOF0 : TOF;
    CTU0 : CTU;
    Val1 : USINT;
    Val2 : USINT;
    Val3 : USINT;
    Val4 : USINT;
    Val5 : USINT;
    _TMP_GT3_OUT : BOOL;
    R_TRIG1 : R_TRIG;
  END_VAR

  _TMP_GT3_OUT := GT(Ana0, 400);
  Out2 := _TMP_GT3_OUT;
  Out0 := Inp0;
  TON0(IN := NOT(Out3), PT := T#480ms);
  TOF0(IN := TON0.Q, PT := T#480ms);
  Out3 := TOF0.Q;
  Out1 := Inp1;
  Out4 := Inp4;
  Out5 := Inp5;
  R_TRIG1(CLK := Out3);
  CTU0(CU := R_TRIG1.Q, R := Cout, PV := 20);
  Cval0 := CTU0.CV;
  Cout := CTU0.Q;
  Out6 := Inp6;
  Out7 := Inp7;
END_PROGRAM

CONFIGURATION Config0

  RESOURCE Res0 ON PLC
    TASK task0(INTERVAL := T#20ms,PRIORITY := 0);
    PROGRAM instance0 WITH task0 : program0;
  END_RESOURCE
END_CONFIGURATION

(* ---- lb_claude_assisted_eedf635bb135_0019.st ---- *)
PROGRAM basic_ladder
  VAR
    input1 AT %IX0.0 : BOOL := FALSE;
    input2 AT %IX0.1 : BOOL := TRUE;
    output1 AT %QX0.0 : BOOL;
    output2 AT %QX0.1 : BOOL;
    reset AT %IX0.2 : BOOL := FALSE;
  END_VAR
  VAR
    TON0 : TON;
    TOF0 : TOF;
    CTU0 : CTU;
    TP0 : TP;
    R_TRIG1 : R_TRIG;
  END_VAR

  TON0(IN := input1, PT := T#500ms);
  TOF0(IN := TON0.Q, PT := T#500ms);
  output1 := TOF0.Q;
  TP0(IN := input2, PT := T#100ms);
  R_TRIG1(CLK := TP0.Q);
  CTU0(CU := R_TRIG1.Q, R := reset, PV := 7);
  output2 := CTU0.Q;
END_PROGRAM

(* ---- lb_claude_assisted_f8a8074915c6_0020.st ---- *)
PROGRAM program0
  VAR
    S1 : BOOL;
    Actual_Input_Signal : BOOL;
    Cylinder_1 : BOOL;
    Cylinder_2 : BOOL;
    Cylinder_3 : BOOL;
    y : BOOL;
    B2 : BOOL;
    B3 : BOOL;
    Reset : BOOL;
    B4 : BOOL;
    B5 : BOOL;
    B6 : BOOL;
    x : BOOL;
    B7 : BOOL;
    TON0 : TON;
    CTU0 : CTU;
    CTU1 : CTU;
    TOF0 : TOF;
    CTU2 : CTU;
    TON1 : TON;
    _TMP_NOT49_OUT : BOOL;
    _TMP_NOT8_OUT : BOOL;
    _TMP_XOR14_OUT : BOOL;
    _TMP_NOT15_OUT : BOOL;
    _TMP_NOT19_OUT : BOOL;
    _TMP_AND17_OUT : BOOL;
    R_TRIG1 : R_TRIG;
    _TMP_GT24_OUT : BOOL;
    _TMP_NOT48_OUT : BOOL;
    R_TRIG2 : R_TRIG;
    _TMP_GT25_OUT : BOOL;
    _TMP_AND29_OUT : BOOL;
    _TMP_SUB28_OUT : INT;
    _TMP_EQ30_OUT : BOOL;
    _TMP_AND32_OUT : BOOL;
    _TMP_NOT33_OUT : BOOL;
    _TMP_EQ36_OUT : BOOL;
    R_TRIG3 : R_TRIG;
    _TMP_XOR44_OUT : BOOL;
  END_VAR

  Actual_Input_Signal := S1;
  _TMP_NOT49_OUT := NOT(Reset);
  Actual_Input_Signal := _TMP_NOT49_OUT;
  S1 := Actual_Input_Signal;
  B7 := Actual_Input_Signal;
  y := B7;
  _TMP_NOT8_OUT := NOT(y);
  Cylinder_1 := _TMP_NOT8_OUT;
  TON0(IN := B2, PT := T#4s);
  _TMP_XOR14_OUT := XOR(B2, TON0.Q);
  Cylinder_2 := _TMP_XOR14_OUT;
  _TMP_NOT15_OUT := NOT(_TMP_XOR14_OUT);
  _TMP_NOT19_OUT := NOT(B6);
  _TMP_AND17_OUT := AND(_TMP_NOT15_OUT, TON0.Q, _TMP_NOT19_OUT);
  Cylinder_3 := _TMP_AND17_OUT;
  R_TRIG1(CLK := Cylinder_3);
  CTU0(CU := R_TRIG1.Q, R := S1, PV := 10);
  _TMP_GT24_OUT := GT(CTU0.CV, 0);
  _TMP_NOT48_OUT := NOT(Cylinder_3);
  R_TRIG2(CLK := _TMP_NOT48_OUT);
  CTU1(CU := R_TRIG2.Q, R := S1, PV := 10);
  _TMP_GT25_OUT := GT(CTU1.CV, 0);
  _TMP_AND29_OUT := AND(_TMP_GT24_OUT, _TMP_GT25_OUT);
  _TMP_SUB28_OUT := SUB(CTU0.CV, CTU1.CV);
  _TMP_EQ30_OUT := EQ(_TMP_SUB28_OUT, 0);
  _TMP_AND32_OUT := AND(_TMP_AND29_OUT, _TMP_EQ30_OUT);
  _TMP_NOT33_OUT := NOT(_TMP_AND32_OUT);
  TOF0(IN := _TMP_NOT33_OUT, PT := T#2s);
  _TMP_EQ36_OUT := EQ(_TMP_AND32_OUT, TOF0.Q);
  R_TRIG3(CLK := _TMP_EQ36_OUT);
  CTU2(CU := R_TRIG3.Q, R := S1, PV := 10);
  x := CTU2.Q;
  TON1(IN := x, PT := T#30s);
  _TMP_XOR44_OUT := XOR(x, TON1.Q);
  Reset := _TMP_XOR44_OUT;
  y := _TMP_EQ36_OUT;
END_PROGRAM

CONFIGURATION Config0

  RESOURCE Res0 ON PLC
    TASK task0(INTERVAL := T#20ms,PRIORITY := 0);
    PROGRAM instance0 WITH task0 : program0;
  END_RESOURCE
END_CONFIGURATION

(* ---- lb_e066873262e0_alarm_suppression_assignment_0024.st ---- *)
PROGRAM My_Program
  VAR
    button1 AT %IX0.0 : BOOL;
    button2 AT %IX0.1 : BOOL;
    led AT %QX0.0 : BOOL;
  END_VAR

  VAR
    LED_STATE : BOOL;
    ALARM_STATE: BOOL;
  END_VAR

  LED_STATE := (button1 = button2) AND (button1 = TRUE);
  ALARM_STATE := (button1 = TRUE) AND (button2 = FALSE);
  IF LED_STATE OR ALARM_STATE THEN
    led := TRUE;
  ELSE
    led := FALSE;
  END_IF;
END_PROGRAM

CONFIGURATION STD_CONF

  RESOURCE STD_RESSOURCE ON PLC
    TASK TaskMain(INTERVAL := T#50ms,PRIORITY := 0);
    PROGRAM Inst0 WITH TaskMain : My_Program;
  END_RESOURCE
END_CONFIGURATION
